// Mitsubishi GX Works2 project: 42015018_GX_Works2   PLC: Q00J

PROGRAM MAIN
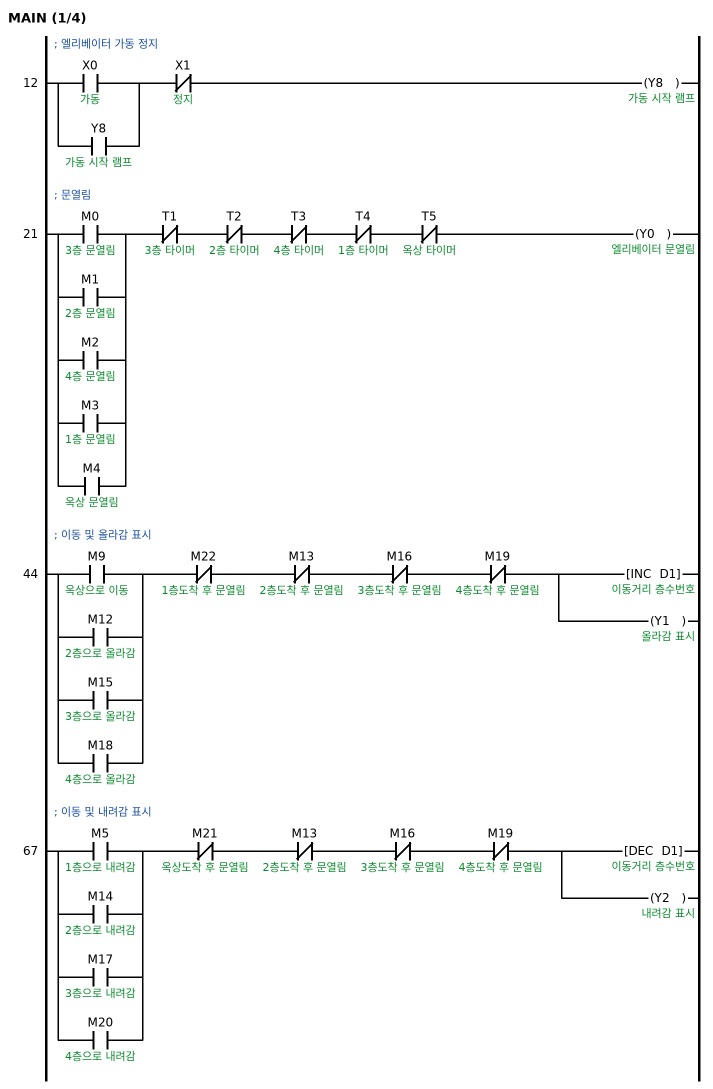
; 엘리베이터 가동 정지
12    LD      X0  ; 가동
      OR      Y8  ; 가동 시작 램프
      ANI     X1  ; 정지
      OUT     Y8  ; 가동 시작 램프
; 문열림
21    LD      M0  ; 3층 문열림
      OR      M1  ; 2층 문열림
      OR      M2  ; 4층 문열림
      OR      M3  ; 1층 문열림
      OR      M4  ; 옥상 문열림
      ANI     T1  ; 3층 타이머
      ANI     T2  ; 2층 타이머
      ANI     T3  ; 4층 타이머
      ANI     T4  ; 1층 타이머
      ANI     T5  ; 옥상 타이머
      OUT     Y0  ; 엘리베이터 문열림
; 이동 및 올라감 표시
44    LD      M9  ; 옥상으로 이동
      OR      M12  ; 2층으로 올라감
      OR      M15  ; 3층으로 올라감
      OR      M18  ; 4층으로 올라감
      ANI     M22  ; 1층도착 후 문열림
      ANI     M13  ; 2층도착 후 문열림
      ANI     M16  ; 3층도착 후 문열림
      ANI     M19  ; 4층도착 후 문열림
      INC     D1  ; 이동거리 층수번호
      OUT     Y1  ; 올라감 표시
; 이동 및 내려감 표시
67    LD      M5  ; 1층으로 내려감
      OR      M14  ; 2층으로 내려감
      OR      M17  ; 3층으로 내려감
      OR      M20  ; 4층으로 내려감
      ANI     M21  ; 옥상도착 후 문열림
      ANI     M13  ; 2층도착 후 문열림
      ANI     M16  ; 3층도착 후 문열림
      ANI     M19  ; 4층도착 후 문열림
      DEC     D1
      OUT     Y2  ; 내려감 표시
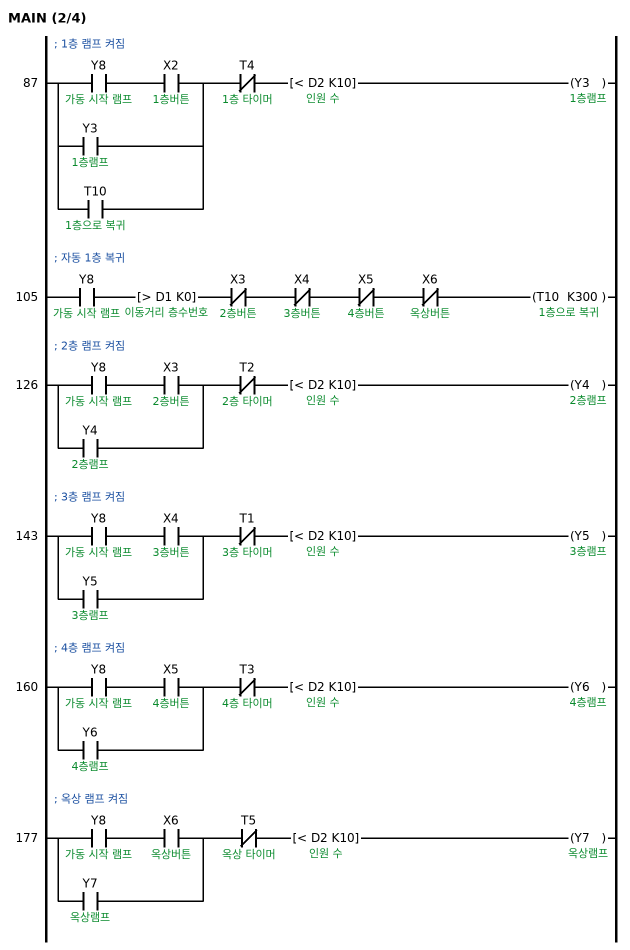
; 1층 램프 켜짐
87    LD      Y8  ; 가동 시작 램프
      AND     X2  ; 1층버튼
      OR      Y3  ; 1층램프
      OR      T10  ; 1층으로 복귀
      ANI     T4  ; 1층 타이머
      AND<    D2 K10  ; 인원 수
      OUT     Y3  ; 1층램프
; 자동 1층 복귀
105   LD      Y8  ; 가동 시작 램프
      AND>    D1 K0  ; 이동거리 층수번호
      ANI     X3  ; 2층버튼
      ANI     X4  ; 3층버튼
      ANI     X5  ; 4층버튼
      ANI     X6  ; 옥상버튼
      OUT     T10 K300  ; 1층으로 복귀
; 2층 램프 켜짐
126   LD      Y8  ; 가동 시작 램프
      AND     X3  ; 2층버튼
      OR      Y4  ; 2층램프
      ANI     T2  ; 2층 타이머
      AND<    D2 K10  ; 인원 수
      OUT     Y4  ; 2층램프
; 3층 램프 켜짐
143   LD      Y8  ; 가동 시작 램프
      AND     X4  ; 3층버튼
      OR      Y5  ; 3층램프
      ANI     T1  ; 3층 타이머
      AND<    D2 K10  ; 인원 수
      OUT     Y5  ; 3층램프
; 4층 램프 켜짐
160   LD      Y8  ; 가동 시작 램프
      AND     X5  ; 4층버튼
      OR      Y6  ; 4층램프
      ANI     T3  ; 4층 타이머
      AND<    D2 K10  ; 인원 수
      OUT     Y6  ; 4층램프
; 옥상 램프 켜짐
177   LD      Y8  ; 가동 시작 램프
      AND     X6  ; 옥상버튼
      OR      Y7  ; 옥상램프
      ANI     T5  ; 옥상 타이머
      AND<    D2 K10  ; 인원 수
      OUT     Y7  ; 옥상램프
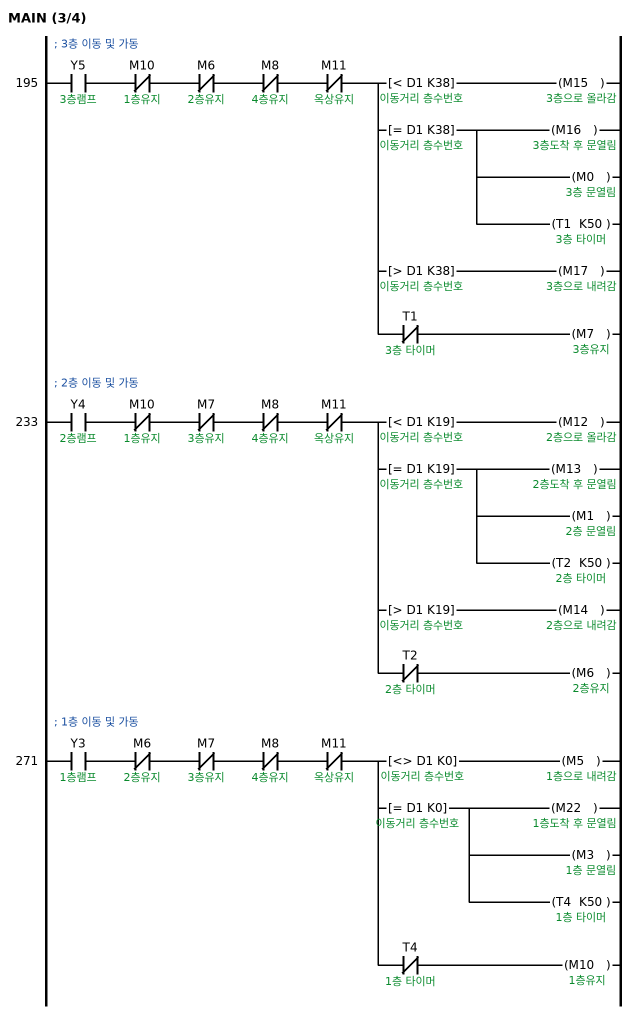
; 3층 이동 및 가동
195   LD      Y5  ; 3층램프
      ANI     M10  ; 1층유지
      ANI     M6  ; 2층유지
      ANI     M8  ; 4층유지
      ANI     M11  ; 옥상유지
      MPS
      AND<    D1 K38  ; 이동거리 층수번호
      OUT     M15  ; 3층으로 올라감
      MRD
      AND=    D1 K38  ; 이동거리 층수번호
      OUT     M16  ; 3층도착 후 문열림
      OUT     M0  ; 3층 문열림
      OUT     T1 K50  ; 3층 타이머
      MRD
      AND>    D1 K38  ; 이동거리 층수번호
      OUT     M17  ; 3층으로 내려감
      MPP
      ANI     T1  ; 3층 타이머
      OUT     M7  ; 3층유지
; 2층 이동 및 가동
233   LD      Y4  ; 2층램프
      ANI     M10  ; 1층유지
      ANI     M7  ; 3층유지
      ANI     M8  ; 4층유지
      ANI     M11  ; 옥상유지
      MPS
      AND<    D1 K19  ; 이동거리 층수번호
      OUT     M12  ; 2층으로 올라감
      MRD
      AND=    D1 K19  ; 이동거리 층수번호
      OUT     M13  ; 2층도착 후 문열림
      OUT     M1  ; 2층 문열림
      OUT     T2 K50  ; 2층 타이머
      MRD
      AND>    D1 K19  ; 이동거리 층수번호
      OUT     M14  ; 2층으로 내려감
      MPP
      ANI     T2  ; 2층 타이머
      OUT     M6  ; 2층유지
; 1층 이동 및 가동
271   LD      Y3  ; 1층램프
      ANI     M6  ; 2층유지
      ANI     M7  ; 3층유지
      ANI     M8  ; 4층유지
      ANI     M11  ; 옥상유지
      MPS
      AND<>   D1 K0  ; 이동거리 층수번호
      OUT     M5  ; 1층으로 내려감
      MRD
      AND=    D1 K0  ; 이동거리 층수번호
      OUT     M22  ; 1층도착 후 문열림
      OUT     M3  ; 1층 문열림
      OUT     T4 K50  ; 1층 타이머
      MPP
      ANI     T4  ; 1층 타이머
      OUT     M10  ; 1층유지
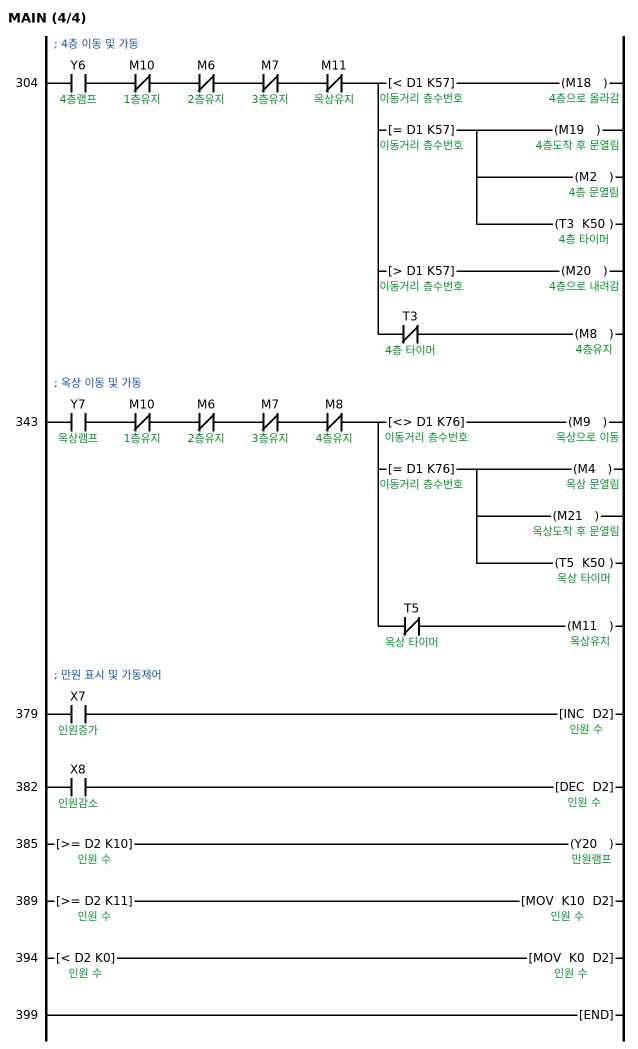
; 4층 이동 및 가동
304   LD      Y6  ; 4층램프
      ANI     M10  ; 1층유지
      ANI     M6  ; 2층유지
      ANI     M7  ; 3층유지
      ANI     M11  ; 옥상유지
      MPS
      AND<    D1 K57  ; 이동거리 층수번호
      OUT     M18  ; 4층으로 올라감
      MRD
      AND=    D1 K57  ; 이동거리 층수번호
      OUT     M19  ; 4층도착 후 문열림
      OUT     M2  ; 4층 문열림
      OUT     T3 K50  ; 4층 타이머
      MRD
      AND>    D1 K57  ; 이동거리 층수번호
      OUT     M20  ; 4층으로 내려감
      MPP
      ANI     T3  ; 4층 타이머
      OUT     M8  ; 4층유지
; 옥상 이동 및 가동
343   LD      Y7  ; 옥상램프
      ANI     M10  ; 1층유지
      ANI     M6  ; 2층유지
      ANI     M7  ; 3층유지
      ANI     M8  ; 4층유지
      MPS
      AND<>   D1 K76  ; 이동거리 층수번호
      OUT     M9  ; 옥상으로 이동
      MRD
      AND=    D1 K76  ; 이동거리 층수번호
      OUT     M4  ; 옥상 문열림
      OUT     M21  ; 옥상도착 후 문열림
      OUT     T5 K50  ; 옥상 타이머
      MPP
      ANI     T5  ; 옥상 타이머
      OUT     M11  ; 옥상유지
; 만원 표시 및 가동제어
379   LD      X7  ; 인원증가
      INC     D2
382   LD      X8  ; 인원감소
      DEC     D2
385   LD>=    D2 K10  ; 인원 수
      OUT     Y20  ; 만원램프
389   LD>=    D2 K11  ; 인원 수
      MOV     K10 D2
394   LD<     D2 K0  ; 인원 수
      MOV     K0 D2
399   END
END_PROGRAM
